SUBAPPLICATION AX_LinksRechts_T_FF (* Links/Rechts Umschaltung mittels Toggle-Flip-Flop (AX-Adapter) *)
  (* Standard: 61499-2; Description: Copyright (c) 2023 Meisterschulen am Ostbahnhof This program and the accompanying materials are made available under the terms of the Eclipse Public License 2.0 which is available at https://www.eclipse.org/legal/epl-2.0/ SPDX-License-Identifier: EPL-2.0 *)
  (* Version 1.0, 2026-01-13, Franz Höpfinger, Meisterschulen am Ostbahnhof, initial API and implementation and/or initial documentation *)
  PACKAGE MyLib::sys;
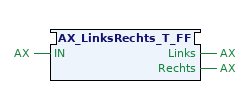
  SOCKETS
    IN : adapter::types::unidirectional::AX;
  END_SOCKETS
  PLUGS
    Links : adapter::types::unidirectional::AX;
    Rechts : adapter::types::unidirectional::AX;
  END_PLUGS
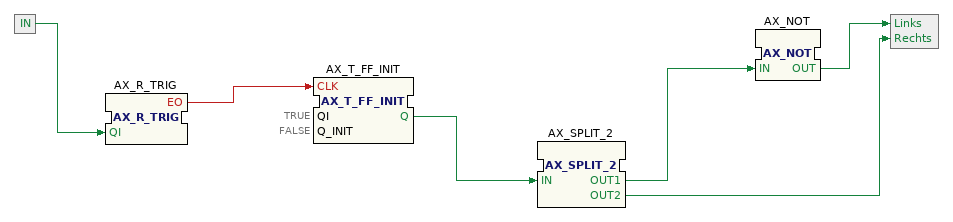
  (* der AX_T_FF_INIT schaltet den Ausgang Aktiv auf FALSE, somit ist LINKS dann TRUE. *)
  FBS
    AX_T_FF_INIT : adapter::events::unidirectional::AX_T_FF_INIT(QI := TRUE, Q_INIT := FALSE);
    AX_R_TRIG : adapter::events::unidirectional::AX_R_TRIG;
    AX_NOT : adapter::booleanOperators::AX_NOT;
    AX_SPLIT_2 : adapter::events::unidirectional::AX_SPLIT_2;
  END_FBS
  EVENT_CONNECTIONS
    AX_R_TRIG.EO TO AX_T_FF_INIT.CLK;
  END_CONNECTIONS
  ADAPTER_CONNECTIONS
    IN TO AX_R_TRIG.QI;
    AX_NOT.OUT TO Links;
    AX_T_FF_INIT.Q TO AX_SPLIT_2.IN;
    AX_SPLIT_2.OUT1 TO AX_NOT.IN;
    AX_SPLIT_2.OUT2 TO Rechts;
  END_CONNECTIONS
END_SUBAPPLICATION
